PROGRAM MAIN
VAR
	fbMachine			:	FB_Machine(3);
	bButton				:	BOOL;
	bInsertCoin			:	BOOL;
	bTakeProduct		:	BOOL;
	bTakeCoin			:	BOOL;
END_VAR

fbMachine(	bButton	:= bButton,
			bInsertCoin := bInsertCoin,
			bTakeProduct := bTakeProduct,
			bTakeCoin := bTakeCoin);	

bButton := FALSE;
bInsertCoin := FALSE;
bTakeProduct := FALSE;
bTakeCoin := FALSE;

END_PROGRAM

(* stored: Version 1.1.0.1, ProductVersion 3.1.4022.12
   POU MAIN: Id {98dd6e6b-9ff3-4f85-9d6c-d1949ebdfc91}, SpecialFunc None *)
